// Mitsubishi GX Works2 project: BookEX6_47 Other   PLC: Q13UDV

// global labels: Global
VAR_GLOBAL
  bVar0 AT M5000 : BOOL;
  abArray0 AT M5010 : ARRAY [0..49] OF BOOL;
  sStr0 AT D5000 : STRING[199];
  sStr1 AT D5100 : STRING[199];
  sStr2 AT D5200 : STRING[199];
  sStr3 AT D5300 : STRING[199];
  sStr4 AT D5400 : STRING[199];
  sStr5 AT D5500 : STRING[199];
  sStr6 AT D5600 : STRING[199];
  sStr7 AT D5700 : STRING[199];
  sStr8 AT D5800 : STRING[199];
  sStr9 AT D5900 : STRING[199];
  iVar0 AT D4500 : INT;
  iVar1 AT D4501 : INT;
  iVar2 AT D4502 : INT;
  iVar3 AT D4503 : INT;
  iVar4 AT D4504 : INT;
  iVar5 AT D4505 : INT;
  iVar6 AT D4506 : INT;
  iVar7 AT D4507 : INT;
  iVar8 AT D4508 : INT;
  iVar9 AT D4509 : INT;
  dVar0 AT D4510 : DINT;
  dVar1 AT D4512 : DINT;
  dVar2 AT D4514 : DINT;
  dVar3 AT D4516 : DINT;
  dVar4 AT D4518 : DINT;
  dVar5 AT D4520 : DINT;
  dVar6 AT D4522 : DINT;
  dVar7 AT D4524 : DINT;
  dVar8 AT D4526 : DINT;
  dVar9 AT D4528 : DINT;
  wVar0 AT D4530 : WORD;
  wVar1 AT D4531 : WORD;
  wVar2 AT D4532 : WORD;
  wVar3 AT D4533 : WORD;
  wVar4 AT D4534 : WORD;
  wVar5 AT D4535 : WORD;
  wVar6 AT D4536 : WORD;
  wVar7 AT D4537 : WORD;
  wVar8 AT D4538 : WORD;
  wVar9 AT D4539 : WORD;
  dwVar0 AT D4540 : DWORD;
  dwVar1 AT D4542 : DWORD;
  dwVar2 AT D4544 : DWORD;
  dwVar3 AT D4546 : DWORD;
  dwVar4 AT D4548 : DWORD;
  dwVar5 AT D4550 : DWORD;
  dwVar6 AT D4552 : DWORD;
  dwVar7 AT D4554 : DWORD;
  dwVar8 AT D4556 : DWORD;
  dwVar9 AT D4558 : DWORD;
  fsVar0 AT D4560 : REAL;
  fsVar1 AT D4562 : REAL;
  fsVar2 AT D4564 : REAL;
  fsVar3 AT D4566 : REAL;
  fsVar4 AT D4568 : REAL;
  fsVar5 AT D4570 : REAL;
  fsVar6 AT D4572 : REAL;
  fsVar7 AT D4574 : REAL;
  fsVar8 AT D4576 : REAL;
  fsVar9 AT D4578 : REAL;
  tTime0 AT D4620 : TIME;
  tTime1 AT D4622 : TIME;
  tTime2 AT D4624 : TIME;
  tTime3 AT D4626 : TIME;
  tTime4 AT D4628 : TIME;
  tTime5 AT D4630 : TIME;
  tTime6 AT D4632 : TIME;
  tTime7 AT D4634 : TIME;
  tTime8 AT D4636 : TIME;
  tTime9 AT D4638 : TIME;
  tTime10 AT D4640 : TIME;
  bVar1 AT M5001 : BOOL;
  bVar2 AT M5002 : BOOL;
  bVar3 AT M5003 : BOOL;
  bVar4 AT M5004 : BOOL;
  bVar5 AT M5005 : BOOL;
  bVar6 AT M5006 : BOOL;
  bVar7 AT M5007 : BOOL;
  bVar8 AT M5008 : BOOL;
  bVar9 AT M5009 : BOOL;
  abArray1 AT M5060 : ARRAY [0..49] OF BOOL;
  abArray2 AT M5110 : ARRAY [0..49] OF BOOL;
  abArray3 AT M5160 : ARRAY [0..49] OF BOOL;
  abArray4 AT M5210 : ARRAY [0..49] OF BOOL;
  abArray5 AT M5260 : ARRAY [0..49] OF BOOL;
  abArray6 AT M5310 : ARRAY [0..49] OF BOOL;
  abArray7 AT M5360 : ARRAY [0..49] OF BOOL;
  abArray8 AT M5410 : ARRAY [0..49] OF BOOL;
  abArray9 AT M5460 : ARRAY [0..49] OF BOOL;
  afsPen0 AT D2000 : ARRAY [0..499] OF REAL;
  afsPen1 AT D3000 : ARRAY [0..499] OF REAL;
END_VAR
// user libraries (not included): HMI

PROGRAM ExADRSET
(* structured ladder/FBD written out as ST: instructions are called as NAME(EN, inputs, outputs); _pN, _eN, _tN stand for wires *)
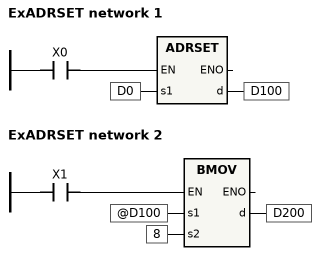
(* network 1 *)
ADRSET(X0, D0, D100);
(* network 2 *)
BMOV(X1, @D100, 8, D200);
END_PROGRAM

PROGRAM ExKEY
(* structured ladder/FBD written out as ST: instructions are called as NAME(EN, inputs, outputs); _pN, _eN, _tN stand for wires *)
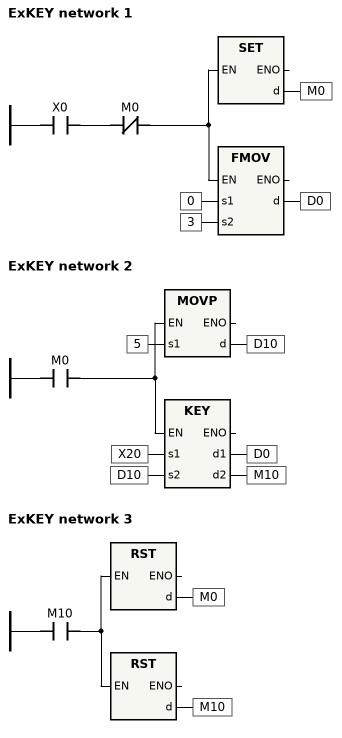
(* network 1 *)
_p1 := X0 AND NOT M0;
SET(_p1, M0);
FMOV(_p1, 0, 3, D0);
(* network 2 *)
MOVP(M0, 5, D10);
KEY(M0, X20, D10, D0, M10);
(* network 3 *)
RST(M10, M0);
RST(M10, M10);
END_PROGRAM

PROGRAM ExDEV
VAR
  Mov4INT_1 : Mov4INT;
END_VAR
(* structured ladder/FBD written out as ST: instructions are called as NAME(EN, inputs, outputs); _pN, _eN, _tN stand for wires *)
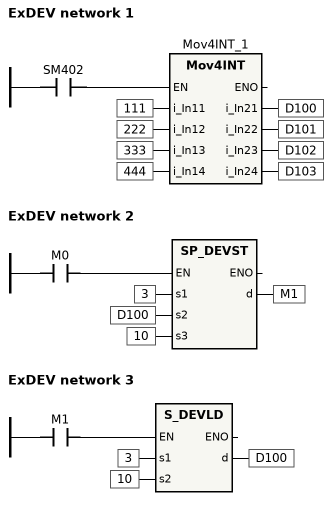
(* network 1 *)
Mov4INT_1(EN := SM402, i_In11 := 111, i_In12 := 222, i_In13 := 333, i_In14 := 444, i_In21 => D100, i_In22 => D101, i_In23 => D102, i_In24 => D103);
(* network 2 *)
SP_DEVST(M0, 3, D100, 10, M1);
(* network 3 *)
S_DEVLD(M1, 3, 10, D100);
END_PROGRAM

PROGRAM ExDUTY
VAR
  HMI05_1 : HMI05;
  ScanOsc_1 : ScanOsc;
  sysScanTime_1 : sysScanTime;
END_VAR
(* structured ladder/FBD written out as ST: instructions are called as NAME(EN, inputs, outputs); _pN, _eN, _tN stand for wires *)
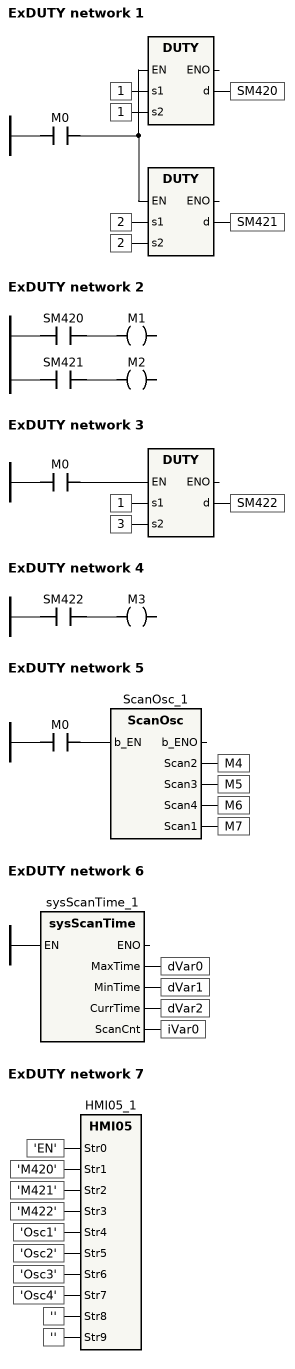
(* network 1 *)
DUTY(M0, 1, 1, SM420);
DUTY(M0, 2, 2, SM421);
(* network 2 *)
M1 := SM420;
M2 := SM421;
(* network 3 *)
DUTY(M0, 1, 3, SM422);
(* network 4 *)
M3 := SM422;
(* network 5 *)
ScanOsc_1(b_EN := M0, Scan2 => M4, Scan3 => M5, Scan4 => M6, Scan1 => M7);
(* network 6 *)
sysScanTime_1(EN := TRUE, MaxTime => dVar0, MinTime => dVar1, CurrTime => dVar2, ScanCnt => iVar0);
(* network 7 *)
HMI05_1(Str0 := 'EN', Str1 := 'M420', Str2 := 'M421', Str3 := 'M422', Str4 := 'Osc1', Str5 := 'Osc2', Str6 := 'Osc3', Str7 := 'Osc4', Str8 := '', Str9 := '');
END_PROGRAM

PROGRAM ExFREAD
VAR
  awCtrl : ARRAY [0..7] OF WORD;
  awData : ARRAY [0..9] OF WORD;
  abComp1 : ARRAY [0..1] OF BOOL;
  abComp2 : ARRAY [0..1] OF BOOL;
  Mov4WORD_1 : Mov4WORD;
  Mov4WORD_2 : Mov4WORD;
END_VAR
(* structured ladder/FBD written out as ST: instructions are called as NAME(EN, inputs, outputs); _pN, _eN, _tN stand for wires *)
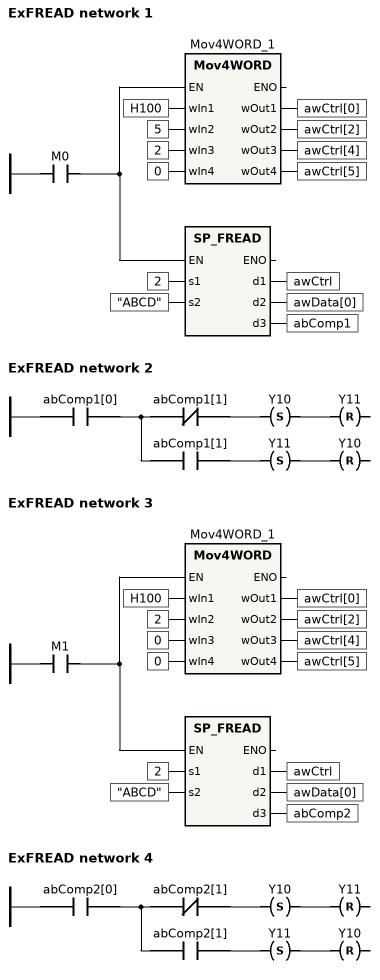
(* network 1 *)
Mov4WORD_1(EN := M0, wIn1 := H100, wIn2 := 5, wIn3 := 2, wIn4 := 0, wOut1 => awCtrl[0], wOut2 => awCtrl[2], wOut3 => awCtrl[4], wOut4 => awCtrl[5]);
SP_FREAD(M0, 2, "ABCD", awCtrl, awData[0], abComp1);
(* network 2 *)
_p1 := abComp1[0] AND NOT abComp1[1];
SET(_p1, Y10);
RST(_p1, Y11);
_p2 := abComp1[0] AND abComp1[1];
SET(_p2, Y11);
RST(_p2, Y10);
(* network 3 *)
Mov4WORD_1(EN := M1, wIn1 := H100, wIn2 := 2, wIn3 := 0, wIn4 := 0, wOut1 => awCtrl[0], wOut2 => awCtrl[2], wOut3 => awCtrl[4], wOut4 => awCtrl[5]);
SP_FREAD(M1, 2, "ABCD", awCtrl, awData[0], abComp2);
(* network 4 *)
_p1 := abComp2[0] AND NOT abComp2[1];
SET(_p1, Y10);
RST(_p1, Y11);
_p2 := abComp2[0] AND abComp2[1];
SET(_p2, Y11);
RST(_p2, Y10);
END_PROGRAM

PROGRAM ExFWRITE
VAR
  awCtrl : ARRAY [0..7] OF WORD;
  awData : ARRAY [0..9] OF WORD;
  abComp1 : ARRAY [0..1] OF BOOL;
  abComp2 : ARRAY [0..1] OF BOOL;
  Mov4WORD_1 : Mov4WORD;
  Mov4WORD_2 : Mov4WORD;
END_VAR
(* structured ladder/FBD written out as ST: instructions are called as NAME(EN, inputs, outputs); _pN, _eN, _tN stand for wires *)
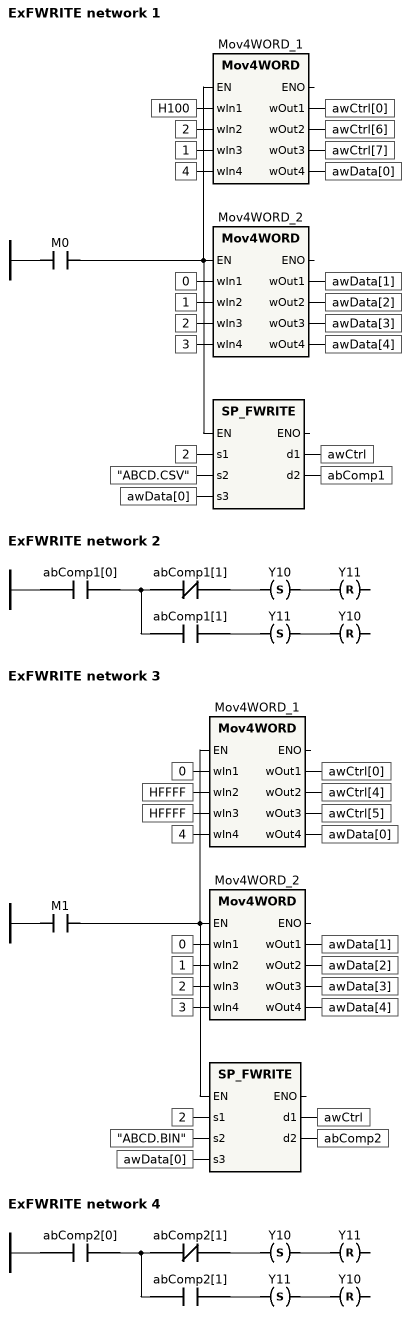
(* network 1 *)
Mov4WORD_1(EN := M0, wIn1 := H100, wIn2 := 2, wIn3 := 1, wIn4 := 4, wOut1 => awCtrl[0], wOut2 => awCtrl[6], wOut3 => awCtrl[7], wOut4 => awData[0]);
Mov4WORD_2(EN := M0, wIn1 := 0, wIn2 := 1, wIn3 := 2, wIn4 := 3, wOut1 => awData[1], wOut2 => awData[2], wOut3 => awData[3], wOut4 => awData[4]);
SP_FWRITE(M0, 2, "ABCD.CSV", awData[0], awCtrl, abComp1);
(* network 2 *)
_p1 := abComp1[0] AND NOT abComp1[1];
SET(_p1, Y10);
RST(_p1, Y11);
_p2 := abComp1[0] AND abComp1[1];
SET(_p2, Y11);
RST(_p2, Y10);
(* network 3 *)
Mov4WORD_1(EN := M1, wIn1 := 0, wIn2 := HFFFF, wIn3 := HFFFF, wIn4 := 4, wOut1 => awCtrl[0], wOut2 => awCtrl[4], wOut3 => awCtrl[5], wOut4 => awData[0]);
Mov4WORD_2(EN := M1, wIn1 := 0, wIn2 := 1, wIn3 := 2, wIn4 := 3, wOut1 => awData[1], wOut2 => awData[2], wOut3 => awData[3], wOut4 => awData[4]);
SP_FWRITE(M1, 2, "ABCD.BIN", awData[0], awCtrl, abComp2);
(* network 4 *)
_p1 := abComp2[0] AND NOT abComp2[1];
SET(_p1, Y10);
RST(_p1, Y11);
_p2 := abComp2[0] AND abComp2[1];
SET(_p2, Y11);
RST(_p2, Y10);
END_PROGRAM

PROGRAM ExRBMOV
VAR
  Mov4WORD_1 : Mov4WORD;
END_VAR
(* structured ladder/FBD written out as ST: instructions are called as NAME(EN, inputs, outputs); _pN, _eN, _tN stand for wires *)
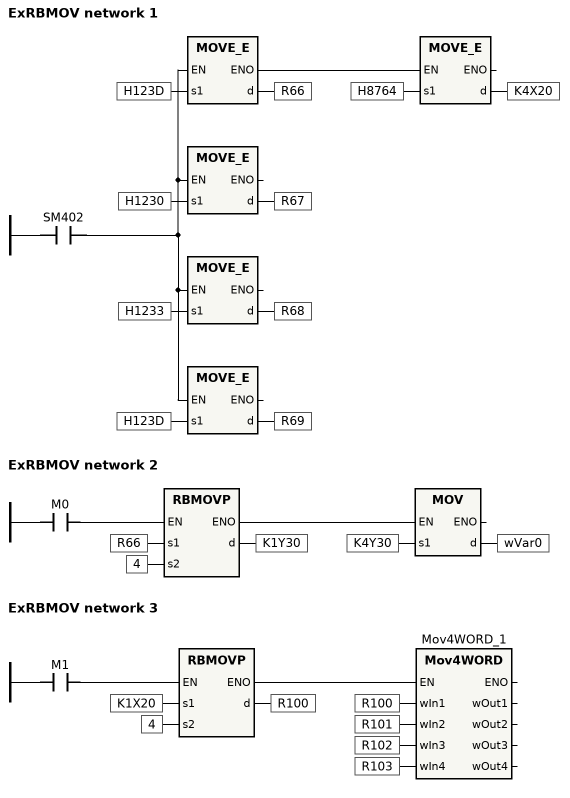
(* network 1 *)
_e1 := MOVE_E(SM402, H123D, R66);
MOVE_E(_e1, H8764, K4X20);
MOVE_E(SM402, H1230, R67);
MOVE_E(SM402, H1233, R68);
MOVE_E(SM402, H123D, R69);
(* network 2 *)
_e1 := RBMOVP(M0, R66, 4, K1Y30);
MOV(_e1, K4Y30, wVar0);
(* network 3 *)
_e1 := RBMOVP(M1, K1X20, 4, R100);
Mov4WORD_1(EN := _e1, wIn1 := R100, wIn2 := R101, wIn3 := R102, wIn4 := R103);
END_PROGRAM

PROGRAM ExTIMCHK
VAR
  HMI05_1 : HMI05;
  HMI03_1 : HMI03;
  newTIMCHK_1 : newTIMCHK;
END_VAR
(* structured ladder/FBD written out as ST: instructions are called as NAME(EN, inputs, outputs); _pN, _eN, _tN stand for wires *)
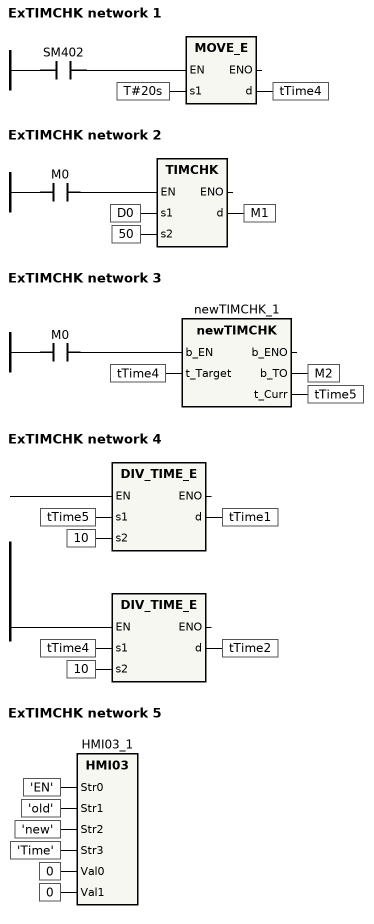
(* network 1 *)
MOVE_E(SM402, T#20s, tTime4);
(* network 2 *)
TIMCHK(M0, D0, 50, M1);
(* network 3 *)
newTIMCHK_1(b_EN := M0, t_Target := tTime4, b_TO => M2, t_Curr => tTime5);
(* network 4 *)
DIV_TIME_E(TRUE, tTime5, 10, tTime1);
DIV_TIME_E(TRUE, tTime4, 10, tTime2);
(* network 5 *)
HMI03_1(Str0 := 'EN', Str1 := 'old', Str2 := 'new', Str3 := 'Time', Val0 := 0, Val1 := 0);
END_PROGRAM

PROGRAM ExTRACE
VAR
  TON_E_1 : TON_E;
  TON_1 : TON;
END_VAR
(* structured ladder/FBD written out as ST: instructions are called as NAME(EN, inputs, outputs); _pN, _eN, _tN stand for wires *)
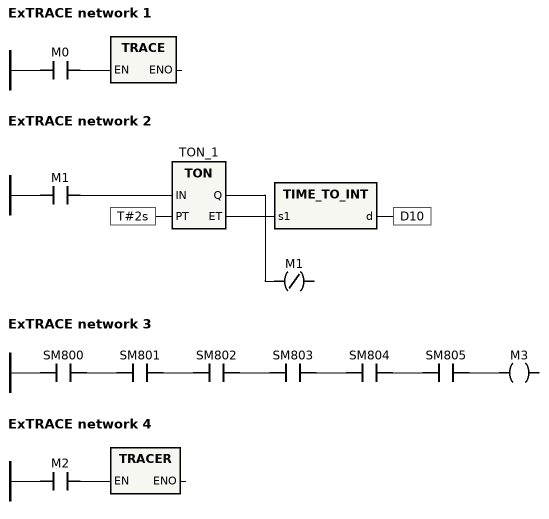
(* network 1 *)
TRACE(M0);
(* network 2 *)
TON_1(IN := M1, PT := T#2s);
M1 := NOT TON_1.Q;
D10 := TIME_TO_INT(TON_1.ET);
(* network 3 *)
M3 := SM800 AND SM801 AND SM802 AND SM803 AND SM804 AND SM805;
(* network 4 *)
TRACER(M2);
END_PROGRAM

PROGRAM ExTYPERD
(* structured ladder/FBD written out as ST: instructions are called as NAME(EN, inputs, outputs); _pN, _eN, _tN stand for wires *)
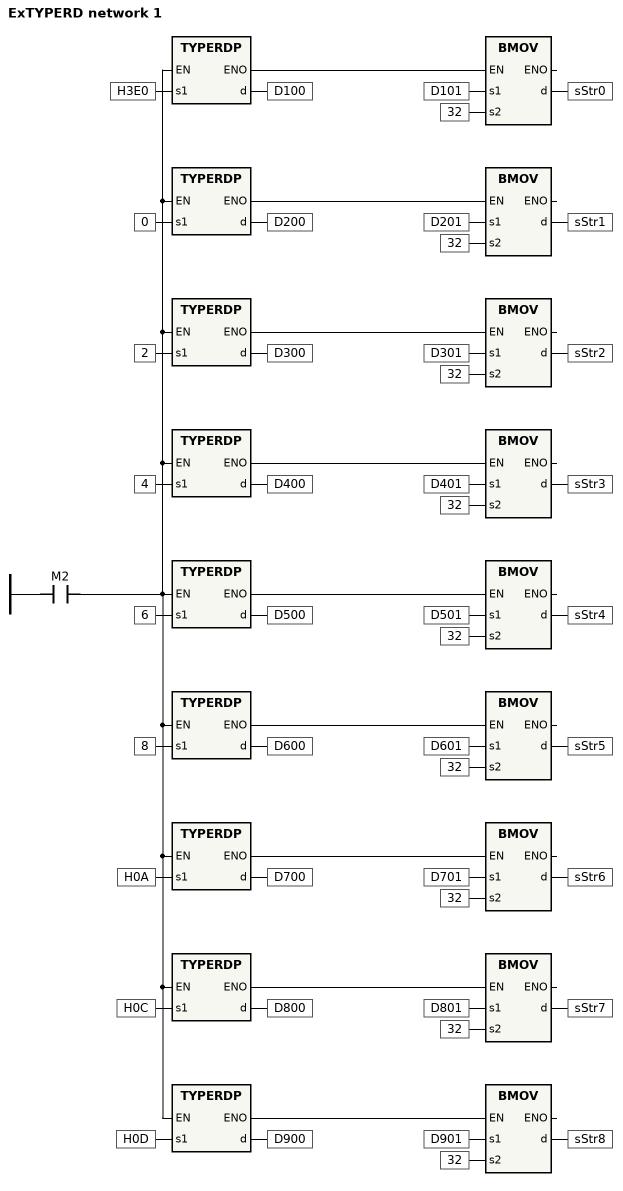
(* network 1 *)
_e1 := TYPERDP(M2, H3E0, D100);
BMOV(_e1, D101, 32, sStr0);
_e2 := TYPERDP(M2, 0, D200);
BMOV(_e2, D201, 32, sStr1);
_e3 := TYPERDP(M2, 2, D300);
BMOV(_e3, D301, 32, sStr2);
_e4 := TYPERDP(M2, 4, D400);
BMOV(_e4, D401, 32, sStr3);
_e5 := TYPERDP(M2, 6, D500);
BMOV(_e5, D501, 32, sStr4);
_e6 := TYPERDP(M2, 8, D600);
BMOV(_e6, D601, 32, sStr5);
_e7 := TYPERDP(M2, H0A, D700);
BMOV(_e7, D701, 32, sStr6);
_e8 := TYPERDP(M2, H0C, D800);
BMOV(_e8, D801, 32, sStr7);
_e9 := TYPERDP(M2, H0D, D900);
BMOV(_e9, D901, 32, sStr8);
END_PROGRAM

PROGRAM ExUNIRD
(* structured ladder/FBD written out as ST: instructions are called as NAME(EN, inputs, outputs); _pN, _eN, _tN stand for wires *)
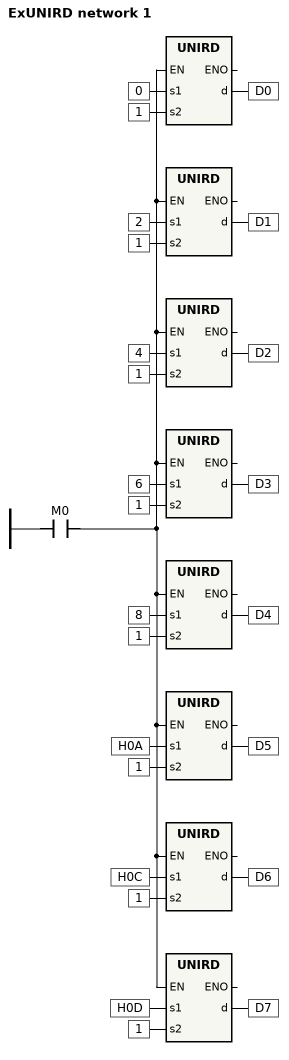
(* network 1 *)
UNIRD(M0, 0, 1, D0);
UNIRD(M0, 2, 1, D1);
UNIRD(M0, 4, 1, D2);
UNIRD(M0, 6, 1, D3);
UNIRD(M0, 8, 1, D4);
UNIRD(M0, H0A, 1, D5);
UNIRD(M0, H0C, 1, D6);
UNIRD(M0, H0D, 1, D7);
END_PROGRAM

PROGRAM ExWDT
(* structured ladder/FBD written out as ST: instructions are called as NAME(EN, inputs, outputs); _pN, _eN, _tN stand for wires *)
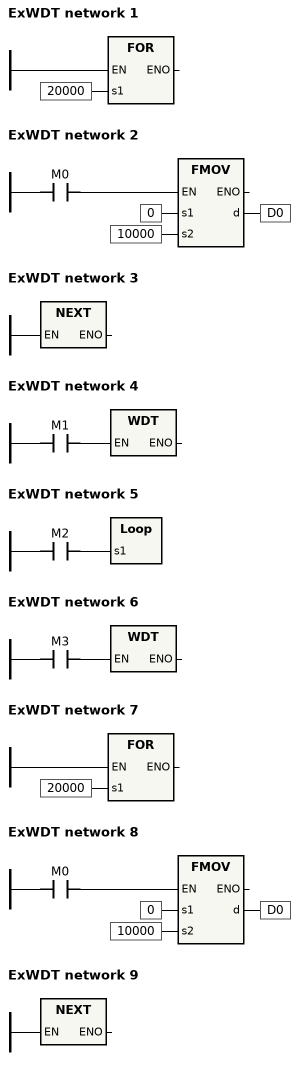
(* network 1 Loop: *)
FOR(TRUE, 20000);
(* network 2 *)
FMOV(M0, 0, 10000, D0);
(* network 3 *)
NEXT(TRUE);
(* network 4 *)
WDT(M1);
(* network 5 *)
(* element kind 9 Loop <- M2 *)
(* network 6 *)
WDT(M3);
(* network 7 *)
FOR(TRUE, 20000);
(* network 8 *)
FMOV(M0, 0, 10000, D0);
(* network 9 *)
NEXT(TRUE);
END_PROGRAM

PROGRAM ExZPush
VAR
  exPushPop_1 : exPushPop;
END_VAR
(* structured ladder/FBD written out as ST: instructions are called as NAME(EN, inputs, outputs); _pN, _eN, _tN stand for wires *)
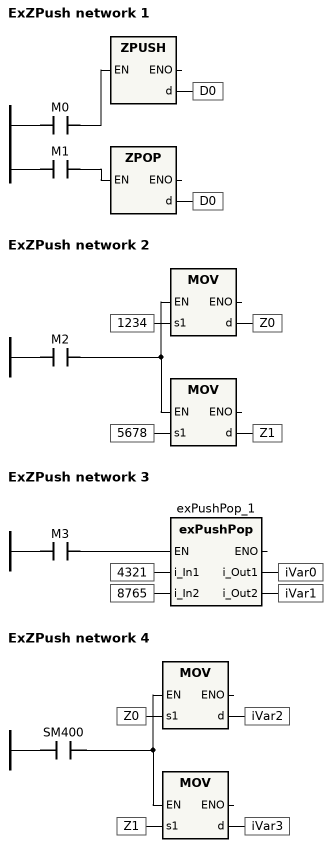
(* network 1 *)
ZPUSH(M0, D0);
ZPOP(M1, D0);
(* network 2 *)
MOV(M2, 1234, Z0);
MOV(M2, 5678, Z1);
(* network 3 *)
exPushPop_1(EN := M3, i_In1 := 4321, i_In2 := 8765, i_Out1 => iVar0, i_Out2 => iVar1);
(* network 4 *)
MOV(SM400, Z0, iVar2);
MOV(SM400, Z1, iVar3);
END_PROGRAM

PROGRAM ExZR
(* structured ladder/FBD written out as ST: instructions are called as NAME(EN, inputs, outputs); _pN, _eN, _tN stand for wires *)
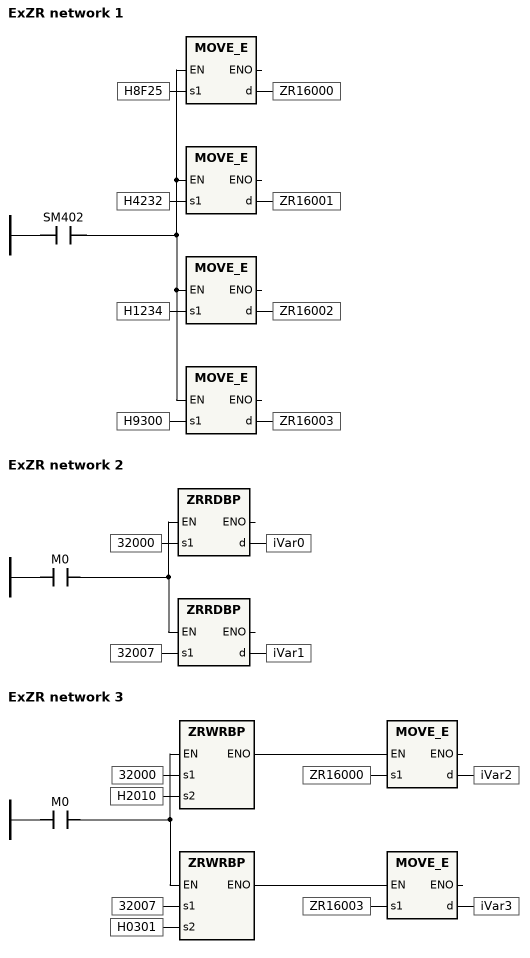
(* network 1 *)
MOVE_E(SM402, H8F25, ZR16000);
MOVE_E(SM402, H4232, ZR16001);
MOVE_E(SM402, H1234, ZR16002);
MOVE_E(SM402, H9300, ZR16003);
(* network 2 *)
ZRRDBP(M0, 32000, iVar0);
ZRRDBP(M0, 32007, iVar1);
(* network 3 *)
_e1 := ZRWRBP(M0, 32000, H2010);
MOVE_E(_e1, ZR16000, iVar2);
_e2 := ZRWRBP(M0, 32007, H0301);
MOVE_E(_e2, ZR16003, iVar3);
END_PROGRAM

FUNCTION_BLOCK exPushPop
VAR_INPUT
  i_In1 : INT;
  i_In2 : INT;
END_VAR
VAR_OUTPUT
  i_Out1 : INT;
  i_Out2 : INT;
END_VAR
VAR
  aiSaveZ1 : ARRAY [0..41] OF INT;
  aiSaveZ2 : ARRAY [0..20] OF INT;
END_VAR
(* 인덱스 레지스터 저장 *)
ZPUSH(TRUE, aiSaveZ1[0]);
(* FB내 인덱스 레지스터사용*)
	Z0 := i_In1;
	(* 인덱스 레지스터 저장 *)
	ZPUSH(TRUE, aiSaveZ1[0]);
		Z0 := Z0+1;
		i_Out1 := Z0;
	(* 인덱스 레지스터 복귀 *)
	ZPOP(TRUE, aiSaveZ1[0]);
	Z0 := Z0+2;
	i_Out2 := Z0;
(* 인덱스 레지스터 복귀 *)
ZPOP(TRUE, aiSaveZ1[0]);
END_FUNCTION_BLOCK

FUNCTION_BLOCK newKEY
VAR_INPUT
  b_EN : BOOL;
  ab_Key : ARRAY [0..15] OF BOOL;
END_VAR
VAR_OUTPUT
  b_ENO : BOOL;
  d_Val : DINT;
  dw_Val : DWORD;
END_VAR
VAR
  iPhs : INT;
  ix : INT;
  iy : INT;
  iCnt : INT;
  dwBuff : DWORD;
  dwBuff2 : DWORD;
END_VAR
VAR_OUTPUT
  i_Cnt : INT;
END_VAR
VAR
  iVal : INT;
END_VAR
;
IF NOT b_EN  THEN
	b_ENO := FALSE;
	iCnt := 0;
	dwBuff := 0;
	RETURN;
END_IF;
FOR ix := 1 TO 16 DO 
	IF ab_Key[ix-1] THEN
		EXIT;
	END_IF;
END_FOR;
IF ix = 17 THEN	iy := 0; ELSE iy := ix; END_IF;
IF iy = iPhs OR iy = 0 OR (iCnt > 7 AND iy <> 16) THEN 
	iPhs := iy;
	RETURN;
END_IF;
iPhs := ix;
CASE iPhs OF
	1 : (* +00 *)
			IF iCnt < 7 THEN
				DROL(TRUE, 8, dwBuff);
				dwBuff := dwBuff AND HFFFFFF00;
				iCnt := iCnt + 2;
			END_IF;
	2, 3 : (* 0 *)
			DROL(TRUE, 4, dwBuff);
			dwBuff := dwBuff AND HFFFFFFF0;
			iCnt := iCnt + 1;
	4 : (* Ent *)
			b_ENO := TRUE;
	5..7 : (* 1,2,3 *)
			dwBuff2 := INT_TO_DWORD(iPhs - 4);
			DROL(TRUE, 4, dwBuff);
			dwBuff := dwBuff AND HFFFFFFF0;
			dwBuff := dwBuff OR dwBuff2;
			iCnt := iCnt + 1;
	9..11 : (* 4,5,6 *)
			dwBuff2 := INT_TO_DWORD(iPhs - 5);
			DROL(TRUE, 4, dwBuff);
			dwBuff := dwBuff AND HFFFFFFF0;
			dwBuff := dwBuff OR dwBuff2;
			iCnt := iCnt + 1;
	13..15 : (* 7,8,9 *)
			dwBuff2 := INT_TO_DWORD(iPhs - 6);
			DROL(TRUE, 4, dwBuff);
			dwBuff := dwBuff AND HFFFFFFF0;
			dwBuff := dwBuff OR dwBuff2;
			iCnt := iCnt + 1;
	12 : (* Clear *)
			b_ENO := FALSE;
			iCnt := 0;
			dwBuff := 0;
	16 : (* Back *)
			IF iCnt <> 0 THEN
				DROR(TRUE, 4, dwBuff);
				dwBuff := dwBuff AND H0FFFFFFF;
				iCnt := iCnt - 1;
			END_IF;	
END_CASE;
d_Val := BCD_TO_DINT(dwBuff);
i_Cnt := iCnt;
dw_Val := dwBuff;
END_FUNCTION_BLOCK

FUNCTION_BLOCK newTIMCHK
VAR_INPUT
  b_EN : BOOL;
END_VAR
VAR_OUTPUT
  b_ENO : BOOL;
  b_TO : BOOL;
  t_Curr : TIME;
END_VAR
VAR_INPUT
  t_Target : TIME;
END_VAR
VAR
  TON_1 : TON;
END_VAR
;
b_ENO := b_EN;
IF NOT b_ENO THEN
	TON_1(IN:= FALSE);
	RETURN;
END_IF;	
IF LDP(TRUE, b_EN) THEN
	TON_1(IN:= FALSE);
	b_TO := FALSE;
END_IF;
TON_1(IN:= TRUE, PT:= T#3276700ms);
t_Curr := TON_1.ET;
IF t_Curr >= t_Target THEN
	b_TO := TRUE;
ELSE
	b_TO := FALSE;
END_IF;
END_FUNCTION_BLOCK

FUNCTION_BLOCK ScanOsc
VAR_OUTPUT
  b_ENO : BOOL;
  Scan2 : BOOL;
END_VAR
VAR
  Tmp1 : BOOL;
  Tmp2 : BOOL;
  Tmp3 : BOOL;
  Tmp4 : BOOL;
END_VAR
VAR_OUTPUT
  Scan3 : BOOL;
  Scan4 : BOOL;
  Scan1 : BOOL;
END_VAR
VAR_INPUT
  b_EN : BOOL;
END_VAR
;
b_ENO := b_EN;
IF NOT b_ENO THEN
	Scan1 := FALSE;
	Scan2 := FALSE;
	Scan3 := FALSE;
	Scan4 := FALSE;
	Tmp1 := FALSE;
	Tmp2 := FALSE;
	Tmp3 := FALSE;
	Tmp4 := FALSE;
	RETURN;
END_IF;	
Tmp1 := NOT Tmp1;
Scan1 := Tmp1;
IF LDP(TRUE, Tmp1) THEN
	Tmp2 := NOT Tmp2;
	Scan2 := Tmp2;
END_IF;
IF LDP(TRUE, Tmp2) THEN
	Tmp3 := NOT Tmp3;
	Scan3 := Tmp3;
END_IF;
IF LDP(TRUE, Tmp3) THEN
	Tmp4 := NOT Tmp4;
	Scan4 := Tmp4;
END_IF;
END_FUNCTION_BLOCK

FUNCTION_BLOCK sysScanTime
VAR_OUTPUT
  MaxTime : DINT;
  MinTime : DINT;
  CurrTime : DINT;
  ScanCnt : INT;
END_VAR
VAR
  dTmp1 : DINT;
  dTmp2 : DINT;
END_VAR
;
dTmp1 := INT_TO_DINT(SD520);
dTmp2 := INT_TO_DINT(SD521);
CurrTime := dTmp1*1000+dTmp2;
dTmp1 := INT_TO_DINT(SD524);
dTmp2 := INT_TO_DINT(SD525);
MinTime := dTmp1*1000+dTmp2;
dTmp1 := INT_TO_DINT(SD526);
dTmp2 := INT_TO_DINT(SD527);
MaxTime := dTmp1*1000+dTmp2;
ScanCnt := SD420;
END_FUNCTION_BLOCK

PROGRAM ExETC
VAR
  Mov4INT_1 : Mov4INT;
  Mov4WORD_1 : Mov4WORD;
  Mov4WORD_2 : Mov4WORD;
END_VAR
(* structured ladder/FBD written out as ST: instructions are called as NAME(EN, inputs, outputs); _pN, _eN, _tN stand for wires *)
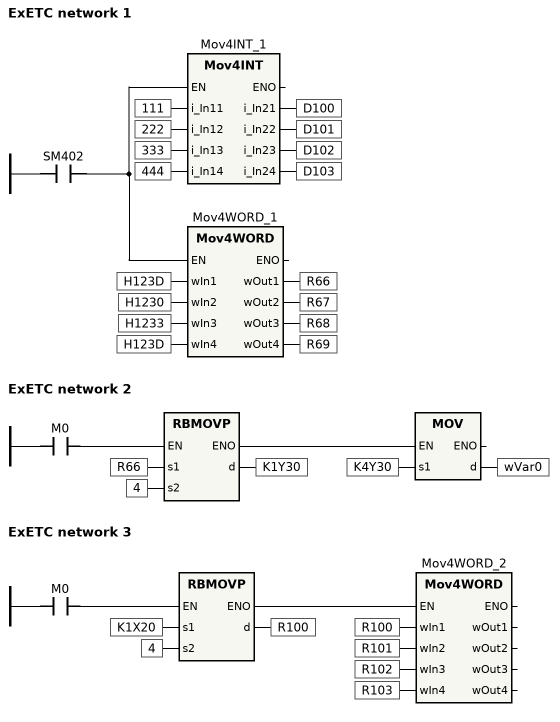
(* network 1 *)
Mov4INT_1(EN := SM402, i_In11 := 111, i_In12 := 222, i_In13 := 333, i_In14 := 444, i_In21 => D100, i_In22 => D101, i_In23 => D102, i_In24 => D103);
Mov4WORD_1(EN := SM402, wIn1 := H123D, wIn2 := H1230, wIn3 := H1233, wIn4 := H123D, wOut1 => R66, wOut2 => R67, wOut3 => R68, wOut4 => R69);
(* network 2 *)
_e1 := RBMOVP(M0, R66, 4, K1Y30);
MOV(_e1, K4Y30, wVar0);
(* network 3 *)
_e1 := RBMOVP(M0, K1X20, 4, R100);
Mov4WORD_2(EN := _e1, wIn1 := R100, wIn2 := R101, wIn3 := R102, wIn4 := R103);
END_PROGRAM
